(* CODESYS project LibraryToInstall.library
   Version: 0.3.1
   Title: MechatronicsCore
   DefaultNamespace: MechatronicsCore
   Placeholder: MechatronicsCore
   Company: Beckhoff Automation LLC

Project tree, tasks and I/O mapping:
  libraries: Core, * (Beckhoff Automation LLC); Tc2_Standard, * (Beckhoff Automation GmbH); Tc2_System, * (Beckhoff Automation GmbH); Tc2_Utilities, * (Beckhoff Automation GmbH)
  _Internal/
    NullObjects/
      Logging/
        function block NullMechatronicsLocalLog [ST]: Clear, Commands, DetailedCommands
        function block NullMechatronicsTracePublisher [ST]: LogMessage, LogMessageInstance, Subscribe, Unsubscribe
    function GetSeverityString [ST]
  Logging/
    Interfaces/
      interface I_ContainMechatronicsLocalLog: CommandLog
      interface I_ContainMechatronicsTracePublisher: TracePublisher
      interface I_MechatronicsLocalLog: Clear, Commands, DetailedCommands
      interface I_MechatronicsLocalLogger
      interface I_MechatronicsLogCommand
      interface I_MechatronicsLogger
      interface I_MechatronicsTracePublisher: Subscribe, Unsubscribe
    function block MechatronicsLocalLogger [ST]: Clear, Commands, DetailedCommands, FB_Init, LogMessage, LogMessageInstance
    function block MechatronicsLogCommand [ST]: Arguments, Message, MessageId, Severity, SourceId, SourceName, TimeStamp
    function block MechatronicsTracePublisher [ST]: LogMessage, LogMessageInstance, Subscribe, Unsubscribe
    global variables TraceParameters
  MoverData/
    Interfaces/
      interface I_ContainMoverData: MoverData
      interface I_MoverData
  Project Information/
    function F_GetCompany [ST]
    function F_GetTitle [ST]
    function F_GetVersion [ST]
  TaskBase/
    Interfaces/
      interface I_TaskResult: TaskName
    function block BaseTaskResult [ST]: Busy, Error, ErrorId, TaskName
  Version/
    global variables Global_Version
*)

// Logging/TraceParameters
{attribute 'qualified_only'}
VAR_GLOBAL CONSTANT
	MAX_NUMBER_LOCAL_LOG   : USINT := 20;
END_VAR

// Version/Global_Version
{attribute 'TcGenerated'}
{attribute 'no-analysis'}
{attribute 'linkalways'}
// This function has been automatically generated from the project information.
VAR_GLOBAL CONSTANT
	{attribute 'const_non_replaced'}
	stLibVersion_MechatronicsCore : ST_LibVersion := (iMajor := 0, iMinor := 3, iBuild := 1, iRevision := 0, nFlags := 0, sVersion := '0.3.1');
END_VAR

// _Internal/NullObjects/Logging/NullMechatronicsLocalLog
{attribute 'conditionalshow'}
{warning disable C0094}
FUNCTION_BLOCK NullMechatronicsLocalLog IMPLEMENTS I_MechatronicsLocalLog
VAR
END_VAR

METHOD Clear
VAR_INPUT
END_VAR
END_METHOD

{attribute 'monitoring':='call'}
PROPERTY Commands : REFERENCE TO ARRAY[0..TraceParameters.MAX_NUMBER_LOCAL_LOG - 1] OF T_MaxString
GET
END_GET
END_PROPERTY

{attribute 'monitoring':='call'}
PROPERTY DetailedCommands : REFERENCE TO ARRAY[0..TraceParameters.MAX_NUMBER_LOCAL_LOG - 1] OF I_MechatronicsLogCommand
GET
END_GET
END_PROPERTY

END_FUNCTION_BLOCK

// Logging/Interfaces/I_MechatronicsLocalLog
INTERFACE I_MechatronicsLocalLog EXTENDS I_Base

METHOD Clear
VAR_INPUT
END_VAR
END_METHOD

{attribute 'monitoring':='call'}
PROPERTY Commands : REFERENCE TO ARRAY[0..TraceParameters.MAX_NUMBER_LOCAL_LOG - 1] OF T_MaxString
GET
END_GET
END_PROPERTY

{attribute 'monitoring':='call'}
PROPERTY DetailedCommands :  REFERENCE TO ARRAY[0..TraceParameters.MAX_NUMBER_LOCAL_LOG - 1] OF I_MechatronicsLogCommand
GET
END_GET
END_PROPERTY

END_INTERFACE

// Logging/Interfaces/I_MechatronicsLogCommand
INTERFACE I_MechatronicsLogCommand EXTENDS I_Base, I_TraceMessageInfo, I_TraceSourceInfo, I_ContainTraceArgument

END_INTERFACE

// _Internal/NullObjects/Logging/NullMechatronicsTracePublisher
{attribute 'conditionalshow'}
{warning disable C0094}
FUNCTION_BLOCK NullMechatronicsTracePublisher IMPLEMENTS I_MechatronicsTracePublisher
VAR
END_VAR

METHOD LogMessage
VAR_INPUT
	Key	: Core.T_MaxString;
	Value	: Core.T_MaxString;
	SourceId	: UDINT := 0;
	TimeStamp	: ULINT := 0;
	MessageId	: UDINT := 1;
	Severity	: USINT := 1;
END_VAR
END_METHOD

METHOD LogMessageInstance
VAR_INPUT
	SourceInfo	: Core.I_TraceSourceInfo;
	MessageInfo	: Core.I_TraceMessageInfo;
	Arguments	: Core.I_TraceArgument := 0;
END_VAR
END_METHOD

METHOD Subscribe
VAR_INPUT
	Logger	: I_MechatronicsLogger;
END_VAR
END_METHOD

METHOD Unsubscribe
VAR_INPUT
	Logger	: I_MechatronicsLogger;
END_VAR
END_METHOD

END_FUNCTION_BLOCK

// Logging/Interfaces/I_MechatronicsTracePublisher
INTERFACE I_MechatronicsTracePublisher EXTENDS I_Base,  I_MechatronicsLogger

METHOD Subscribe
VAR_INPUT
	Logger : I_MechatronicsLogger;
END_VAR
END_METHOD

METHOD Unsubscribe
VAR_INPUT
	Logger : I_MechatronicsLogger;
END_VAR
END_METHOD

END_INTERFACE

// Logging/Interfaces/I_MechatronicsLogger
INTERFACE I_MechatronicsLogger EXTENDS I_TraceLogger,I_TraceInstanceLogger

END_INTERFACE

// _Internal/GetSeverityString
FUNCTION GetSeverityString : T_MaxString
VAR_INPUT
	Severity : USINT;
END_VAR
VAR
END_VAR

CASE Severity OF
	0:
		GetSeverityString := 'Verbose: ';

	1:
		GetSeverityString := 'Info: ';

	2:
		GetSeverityString := 'Warning: ';

	3:
		GetSeverityString := 'Error: ';

	4:
		GetSeverityString := 'Critical Error: ';

ELSE
	GetSeverityString := CONCAT('Severity: ', TO_STRING(Severity));
END_CASE

END_FUNCTION

// Logging/Interfaces/I_ContainMechatronicsLocalLog
INTERFACE I_ContainMechatronicsLocalLog EXTENDS I_Base

{attribute 'monitoring':='call'}
PROPERTY CommandLog : I_MechatronicsLocalLog
GET
END_GET
END_PROPERTY

END_INTERFACE

// Logging/Interfaces/I_ContainMechatronicsTracePublisher
INTERFACE I_ContainMechatronicsTracePublisher EXTENDS I_Base

PROPERTY TracePublisher : I_MechatronicsTracePublisher
GET
END_GET
END_PROPERTY

END_INTERFACE

// Logging/Interfaces/I_MechatronicsLocalLogger
INTERFACE I_MechatronicsLocalLogger EXTENDS I_MechatronicsLocalLog, I_MechatronicsLogger

END_INTERFACE

// Logging/MechatronicsLocalLogger
{attribute 'hide_all_locals'}
FUNCTION_BLOCK MechatronicsLocalLogger IMPLEMENTS I_MechatronicsLocalLogger
VAR
	_LogEntries : ARRAY[0..TraceParameters.MAX_NUMBER_LOCAL_LOG - 1] OF MechatronicsLogCommand;
	_Entries	: ARRAY[0..TraceParameters.MAX_NUMBER_LOCAL_LOG - 1] OF I_MechatronicsLogCommand;
	_SimpleLog	: ARRAY[0..TraceParameters.MAX_NUMBER_LOCAL_LOG - 1] OF T_MaxString;
END_VAR

METHOD Clear
VAR
	i : UDINT;
END_VAR
FOR i := 0 TO TraceParameters.MAX_NUMBER_LOCAL_LOG - 1 DO
	_LogEntries[i].Arguments  := 0;
	_LogEntries[i].Message	  := '';
	_LogEntries[i].MessageId  := 0;
	_LogEntries[i].TimeStamp  := 0;
	_LogEntries[i].SourceId	  := 0;
	_LogEntries[i].SourceName := '';
END_FOR
END_METHOD

{attribute 'monitoring':='call'}
PROPERTY Commands : REFERENCE TO ARRAY[0..TraceParameters.MAX_NUMBER_LOCAL_LOG - 1] OF T_MaxString
GET
Commands REF= _SimpleLog;
END_GET
END_PROPERTY

{attribute 'monitoring':='call'}
PROPERTY DetailedCommands : REFERENCE TO ARRAY[0..TraceParameters.MAX_NUMBER_LOCAL_LOG - 1] OF I_MechatronicsLogCommand
GET
DetailedCommands REF= _Entries;
END_GET
END_PROPERTY

//FB_Init is always available implicitly and it is used primarily for initialization.
//The return value is not evaluated. For a specific influence, you can also declare the
//methods explicitly and provide additional code there with the standard initialization
//code. You can evaluate the return value.
METHOD FB_Init: BOOL
VAR_INPUT
    bInitRetains: BOOL; // TRUE: the retain variables are initialized (reset warm / reset cold)
    bInCopyCode: BOOL;  // TRUE: the instance will be copied to the copy code afterward (online change)   
END_VAR
VAR
	i : UDINT;
END_VAR
FOR i:= 0 TO TraceParameters.MAX_NUMBER_LOCAL_LOG - 1 DO
	_Entries[i] := _LogEntries[i];
END_FOR
END_METHOD

METHOD LogMessage
VAR_INPUT
	Key		  : T_MaxString;
	Value	  : T_MaxString;
	SourceId  : UDINT := 0;
	TimeStamp : ULINT := 0;
	MessageId : UDINT := 1;
	Severity  : USINT := 1;
END_VAR

VAR_INST
	LogSource  : TraceSourceInfo;
	LogMessage : TraceMessageInfo;
END_VAR
LogSource.SourceName := Key;
LogSource.SourceId	 := SourceId;
LogSource.TimeStamp	 := TimeStamp;
LogMessage.Message	 := Value;
LogMessage.MessageId := MessageId;
LogMessage.Severity	 := Severity;
THIS^.LogMessageInstance(LogSource, LogMessage);
END_METHOD

METHOD LogMessageInstance
VAR_INPUT
	SourceInfo	: I_TraceSourceInfo;
	MessageInfo : I_TraceMessageInfo;
	Arguments	: I_TraceArgument := 0;
END_VAR

VAR
	SysTime	 : T_FILETIME64;
	Severity : T_MaxString;
END_VAR
MEMMOVE(ADR(_SimpleLog[1]), ADR(_SimpleLog[0]), SIZEOF(_SimpleLog[0]) * (TraceParameters.MAX_NUMBER_LOCAL_LOG - 1));
MEMMOVE(ADR(_LogEntries[1]), ADR(_LogEntries[0]), SIZEOF(_LogEntries[0]) * (TraceParameters.MAX_NUMBER_LOCAL_LOG - 1));
_LogEntries[0].SourceId	  := SourceInfo.SourceId;
_LogEntries[0].SourceName := SourceInfo.SourceName;
IF SourceInfo.TimeStamp = 0 THEN
	SysTime					 := F_GetSystemTime();
	_LogEntries[0].Timestamp := SysTime;
ELSE
	_LogEntries[0].TimeStamp := SourceInfo.TimeStamp;
END_IF

_LogEntries[0].Message	 := MessageInfo.Message;
_LogEntries[0].MessageId := MessageInfo.MessageId;
_LogEntries[0].Severity	 := MessageInfo.Severity;
_LogEntries[0].Arguments := Arguments;
_SimpleLog[0]			 := CONCAT(SYSTEMTIME_TO_STRING(FILETIME64_TO_SYSTEMTIME(_LogEntries[0].TimeStamp)),
								   CONCAT(' ', CONCAT(GetSeverityString(MessageInfo.Severity), CONCAT(_LogEntries[0].SourceName, CONCAT(': ', _LogEntries[0].Message)))));

IF Arguments <> 0 THEN
	_SimpleLog[0] := CONCAT(_SimpleLog[0], Arguments.ToString());
END_IF
END_METHOD

END_FUNCTION_BLOCK

// Logging/MechatronicsLogCommand
{attribute 'hide_all_locals'}
FUNCTION_BLOCK MechatronicsLogCommand IMPLEMENTS I_MechatronicsLogCommand
VAR
	_MessageInfo : TraceMessageInfo;
	_SourceInfo	 : TraceSourceInfo;
	_Arguments	 : I_TraceArgument;
END_VAR

{attribute 'monitoring' := 'call'}
PROPERTY Arguments : I_TraceArgument
GET
Arguments := _Arguments;
END_GET
SET
_Arguments := Arguments;
END_SET
END_PROPERTY

{attribute 'monitoring':='call'}
PROPERTY Message : T_MaxString
GET
Message := _MessageInfo.Message;
END_GET
SET
_MessageInfo.Message := Message;
END_SET
END_PROPERTY

{attribute 'monitoring':='call'}
PROPERTY MessageId : UDINT
GET
MessageId := _MessageInfo.MessageId;
END_GET
SET
_MessageInfo.MessageId := MessageId;
END_SET
END_PROPERTY

{attribute 'monitoring':='call'}
PROPERTY Severity : USINT
GET
Severity := _MessageInfo.Severity;
END_GET
SET
_MessageInfo.Severity := Severity;
END_SET
END_PROPERTY

{attribute 'monitoring':='call'}
PROPERTY SourceId : UDINT
GET
SourceId := _SourceInfo.SourceId;
END_GET
SET
_SourceInfo.SourceId := SourceId;
END_SET
END_PROPERTY

{attribute 'monitoring':='call'}
PROPERTY SourceName : T_MaxString
GET
SourceName := _SourceInfo.SourceName;
END_GET
SET
_SourceInfo.SourceName := SourceName;
END_SET
END_PROPERTY

{attribute 'monitoring':='call'}
PROPERTY TimeStamp : ULINT
GET
TimeStamp := _SourceInfo.TimeStamp;
END_GET
SET
_SourceInfo.TimeStamp := TimeStamp;
END_SET
END_PROPERTY

END_FUNCTION_BLOCK

// Logging/MechatronicsTracePublisher
FUNCTION_BLOCK MechatronicsTracePublisher IMPLEMENTS I_MechatronicsTracePublisher
VAR
	{attribute 'hide'}
	_Subscribers : Collection;
END_VAR

METHOD LogMessage
VAR_INPUT
	Key		  : T_MaxString;
	Value	  : T_MaxString;
	SourceId  : UDINT := 0;
	TimeStamp : ULINT := 0;
	MessageId : UDINT := 1;
	Severity  : USINT := 1;
END_VAR

VAR
	Logger : I_TraceLogger;
END_VAR
_Subscribers.ResetIterator();
WHILE _Subscribers.MoveToNext DO
	__QUERYINTERFACE(_Subscribers.Current, Logger);
	IF Logger <> 0 THEN
		Logger.LogMessage(Key,
						  Value,
						  SourceId,
						  TimeStamp,
						  MessageId,
						  Severity);
	END_IF
END_WHILE
END_METHOD

METHOD LogMessageInstance
VAR_INPUT
	SourceInfo	: I_TraceSourceInfo;
	MessageInfo : I_TraceMessageInfo;
	Arguments	: I_TraceArgument := 0;
END_VAR

VAR
	Logger : I_TraceInstanceLogger;
END_VAR
_Subscribers.ResetIterator();
WHILE _Subscribers.MoveToNext DO
	__QUERYINTERFACE(_Subscribers.Current, Logger);
	IF Logger <> 0 THEN
		Logger.LogMessageInstance(SourceInfo, MessageInfo, Arguments);
	END_IF
END_WHILE
END_METHOD

METHOD Subscribe
VAR_INPUT
	Logger : I_MechatronicsLogger;
END_VAR
_Subscribers.AddItem(Logger);
END_METHOD

METHOD Unsubscribe
VAR_INPUT
	Logger : I_MechatronicsLogger;
END_VAR
_Subscribers.RemoveItem(Logger);
END_METHOD

END_FUNCTION_BLOCK

// MoverData/Interfaces/I_ContainMoverData
INTERFACE I_ContainMoverData EXTENDS I_Base

{attribute 'monitoring':='call'}
PROPERTY MoverData : I_MoverData
GET
END_GET
SET
END_SET
END_PROPERTY

END_INTERFACE

// MoverData/Interfaces/I_MoverData
INTERFACE I_MoverData EXTENDS I_Base

END_INTERFACE

// Project Information/F_GetCompany
// This function has been automatically generated from the project information.
{attribute 'signature_flag' := '1073741824'}
{attribute 'TcGenerated'}
{attribute 'no-analysis'}
FUNCTION F_GetCompany : WSTRING
VAR_INPUT
	
END_VAR

F_GetCompany := "Beckhoff Automation LLC";

END_FUNCTION

// Project Information/F_GetTitle
// This function has been automatically generated from the project information.
{attribute 'signature_flag' := '1073741824'}
{attribute 'TcGenerated'}
{attribute 'no-analysis'}
FUNCTION F_GetTitle : WSTRING
VAR_INPUT
	
END_VAR

F_GetTitle := "MechatronicsCore";

END_FUNCTION

// Project Information/F_GetVersion
// This function has been automatically generated from the project information.
{attribute 'signature_flag' := '1073741824'}
{attribute 'TcGenerated'}
{attribute 'no-analysis'}
FUNCTION F_GetVersion : ST_LibVersion
VAR_INPUT
	
END_VAR

F_GetVersion.iMajor := 0;
F_GetVersion.iMinor := 3;
F_GetVersion.iBuild := 1;
F_GetVersion.iRevision := 0;
F_GetVersion.sVersion := '0.3.1';
F_GetVersion.nFlags := 0;

END_FUNCTION

// TaskBase/Interfaces/I_TaskResult
INTERFACE I_TaskResult EXTENDS Core.I_TaskResult

{attribute 'monitoring':='call'}
PROPERTY TaskName : String
GET
END_GET
END_PROPERTY

END_INTERFACE

// TaskBase/BaseTaskResult
{attribute 'hide_all_locals'}
FUNCTION_BLOCK BaseTaskResult IMPLEMENTS I_TaskResult
VAR
	_TaskName : T_MaxString;
	_Busy	 : BOOL;
	_Error	 : BOOL;
	_ErrorId : UDINT;
END_VAR

{attribute 'monitoring' := 'call'}
PROPERTY Busy : BOOL
GET
Busy := _Busy;
END_GET
END_PROPERTY

{attribute 'monitoring' := 'call'}
PROPERTY Error : BOOL
GET
Error := _Error;
END_GET
END_PROPERTY

{attribute 'monitoring' := 'call'}
PROPERTY ErrorId : UDINT
GET
ErrorId := _ErrorId;
END_GET
END_PROPERTY

{attribute 'monitoring':='call'}
PROPERTY TaskName : STRING
GET
TaskName := _TaskName;
END_GET
SET
_TaskName := TaskName;
END_SET
END_PROPERTY

END_FUNCTION_BLOCK
